// TwinCAT 3 PLC project MAIN
// ProgramVersion: 3.1.4022.2
// libraries:
//   Tc2_Standard, * (Beckhoff Automation GmbH)
//   Tc2_System, * (Beckhoff Automation GmbH)
//   Tc3_Module, * (Beckhoff Automation GmbH)
// project tree:
//   / GlobalTextList.TcGTLO, PlcTask.TcTTO, Visualization Manager.TcVMO (not stored)
//   POUs/ MAIN.TcPOU, SFC_Test.TcPOU
//   VISUs/ TC_VISU.TcVIS
// real-time tasks:
//   TASK PlcTask: cycle T#10ms, priority 20, ADS port 350

CONFIGURATION MAIN
    RESOURCE PLC ON TwinCAT3
        TASK PlcTask(INTERVAL := T#10ms, PRIORITY := 20);
        PROGRAM MAIN WITH PlcTask : MAIN;
    END_RESOURCE
END_CONFIGURATION

// ---- POUs/MAIN.TcPOU
PROGRAM MAIN
VAR
END_VAR


SFC_Test();

END_PROGRAM

// ---- POUs/SFC_Test.TcPOU
PROGRAM SFC_Test
VAR
	Step0:SFCStepType;
	Step1:SFCStepType;
	Step2:SFCStepType;
	Step3:SFCStepType;
	Step4:SFCStepType;
	Switch1:BOOL;
	Switch2:BOOL;
	Lamp1:BOOL;
	Lamp2:BOOL;
	Lamp3:BOOL;
	Counter:INT;
	Step0_Counter:INT;
	Step1_Counter:INT;
	
END_VAR

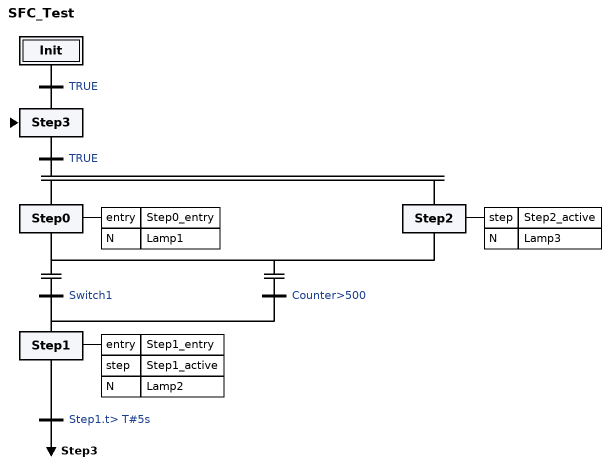
INITIAL_STEP Init:
END_STEP
TRANSITION FROM Init TO Step3
    := TRUE;
END_TRANSITION
STEP Step3:
END_STEP
TRANSITION FROM Step3 TO (Step0, Step2)
    := TRUE;
END_TRANSITION
STEP Step0:
    Step0_entry(P1);  // entry action
    Lamp1(N);
END_STEP
STEP Step2:
    Step2_active(N);  // step action
    Lamp3(N);
END_STEP
TRANSITION FROM (Step0, Step2) TO Step1
    := Switch1;
END_TRANSITION
TRANSITION FROM (Step0, Step2) TO Step1
    := Counter>500;
END_TRANSITION
STEP Step1:
    Step1_entry(P1);  // entry action
    Step1_active(N);  // step action
    Lamp2(N);
END_STEP
TRANSITION FROM Step1 TO Step3
    := Step1.t> T#5s;
END_TRANSITION

ACTION Step0_entry:
Step0_Counter:=500;
END_ACTION

ACTION Step1_active:
Step1_Counter:=Step1_Counter+1;
END_ACTION

ACTION Step1_entry:
Step1_Counter:=0;
Counter:=0;
END_ACTION

ACTION Step2_active:
Counter:=Counter+1;
END_ACTION

ACTION Step4_active:
;
END_ACTION

END_PROGRAM

// ---- VISUs/TC_VISU.TcVIS
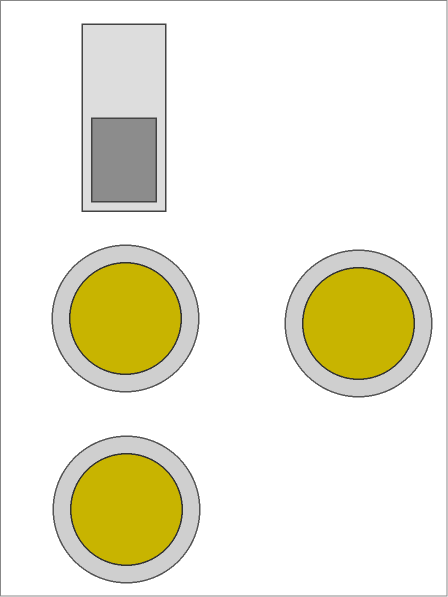
VISUALIZATION TC_VISU  // 448x597
    DipSwitch (30,18 188x199), variable: SFC_Test.Switch1, behaviour: TOGGLE, style: Switch-DipSwitch-Gray
    Lamp1 (38,233 175x171), variable: SFC_Test.Lamp1, style: Lamp-Lamp1-Yellow
    Lamp1 (39,424 175x171), variable: SFC_Test.Lamp2, style: Lamp-Lamp1-Yellow
    Lamp1 (271,238 175x171), variable: SFC_Test.Lamp3, style: Lamp-Lamp1-Yellow
END_VISUALIZATION
